(* Logix 5000 project; controller Oki_4_21_A vendor 1 type 14 code 77 rev 20.11; software revision 20.01 *)

TASK MainTask (continuous, watchdog 500 ms) : MainProgram

MODULES
   Controller : vendor 1 type 14 code 77 (CompactLogixL32EController 0, rev 20.11)
      LocalENB : 1769-L32E Ethernet Port (CompactLogixL32Ethernet 1, rev 20.11)
      Local : CompactBus (CompactVirtualAdapter 3, rev 20.11)
END_MODULES

PROGRAM MainProgram   (* main routine MainRoutine *)

ROUTINE MainRoutine   (* ladder *)
END_ROUTINE
END_PROGRAM
